// TIA Portal V18 export
VAR_GLOBAL   // PLC tag table "03_EL-3"
   "iEL-3" AT %I0.7 : Bool;
   "oEL-3s" AT %Q20.0 : Bool;
   "oEL-3f" AT %Q20.1 : Bool;
END_VAR
